PROGRAM PRG_IM4K2_PPM
VAR
    {attribute 'pytmc' := '
        pv: IM4K2:PPM
        io: io
    '}
     {attribute 'TcLinkTo' := '.fbGige.iIlluminatorINT := TIIB[IM4K2-EL4004-E7]^AO Outputs Channel 1^Analog output;
                              .fbGige.bGigePower := TIIB[IM4K2-EL2004-E3]^Channel 2^Output;
                              .fbPowerMeter.iVoltageINT := TIIB[IM4K2-EL3062-E6]^AI Standard Channel 1^Value;
                              .fbPowerMeter.fbThermoCouple.bError := TIIB[IM4K2-EL3314-E4]^TC Inputs Channel 1^Status^Error;
                              .fbPowerMeter.fbThermoCouple.bUnderrange := TIIB[IM4K2-EL3314-E4]^TC Inputs Channel 1^Status^Underrange;
                              .fbPowerMeter.fbThermoCouple.bOverrange := TIIB[IM4K2-EL3314-E4]^TC Inputs Channel 1^Status^Overrange;
                              .fbPowerMeter.fbThermoCouple.iRaw := TIIB[IM4K2-EL3314-E4]^TC Inputs Channel 1^Value;
                              .fbYagThermoCouple.bError := TIIB[IM4K2-EL3314-E4]^TC Inputs Channel 2^Status^Error;
                              .fbYagThermoCouple.bUnderrange := TIIB[IM4K2-EL3314-E4]^TC Inputs Channel 2^Status^Underrange;
                              .fbYagThermoCouple.bOverrange := TIIB[IM4K2-EL3314-E4]^TC Inputs Channel 2^Status^Overrange;
                              .fbYagThermoCouple.iRaw := TIIB[IM4K2-EL3314-E4]^TC Inputs Channel 2^Value;
                              .fbFlowMeter.iRaw := TIIB[IM1K2-EL3052-E5]^AI Standard Channel 1^Value'}  //IM1/2/3/4K2 same flow meter
    fbIM4K2: FB_PPM;
END_VAR


fbIM4K2.stOut.fPosition := -10.80;
fbIM4K2.stOut.bUseRawCounts := FALSE;
fbIM4K2.stOut.bValid := TRUE;
fbIM4K2.stOut.stPMPS.sPmpsState := 'IM4K2:PPM-OUT';

fbIM4K2.stPower.fPosition := -49.90;
fbIM4K2.stPower.bUseRawCounts := FALSE;
fbIM4K2.stPower.bValid := TRUE;
fbIM4K2.stPower.stPMPS.sPmpsState := 'IM4K2:PPM-POWERMETER';

fbIM4K2.stYag1.fPosition := -73.90;
fbIM4K2.stYag1.bUseRawCounts := FALSE;
fbIM4K2.stYag1.bValid := TRUE;
fbIM4K2.stYag1.stPMPS.sPmpsState := 'IM4K2:PPM-YAG1';

fbIM4K2.stYag2.fPosition := -99.91;
fbIM4K2.stYag2.bUseRawCounts := FALSE;
fbIM4K2.stYag2.bValid := TRUE;
fbIM4K2.stYag2.stPMPS.sPmpsState := 'IM4K2:PPM-YAG2';

fbIM4K2(
    fbArbiter := GVL.fbArbiter2,
    fbFFHWO := GVL.fbFastFaultOutput2,
    stYStage := Main.M8,
    sDeviceName := 'IM4K2:PPM',
    sTransitionKey := 'IM4K2:PPM-TRANSITION',
    bEnableMotion := TRUE,
    bEnableBeamParams := TRUE,
    bEnablePositionLimits := TRUE,
    fFlowOffset := 0.0,
);

END_PROGRAM

(* stored: Version 1.1.0.1, ProductVersion 3.1.4022.18
   POU PRG_IM4K2_PPM: Id {dfd57a27-7901-4447-85ac-e5255b9203c4}, SpecialFunc None *)
